FUNCTION_BLOCK UDINT_Param
VAR_INPUT PERSISTENT
	val			: UDINT;
END_VAR

END_FUNCTION_BLOCK

(* stored: Version 1.1.0.1
   POU UDINT_Param: Id {ad9808ce-25ce-489a-8ce0-4c21fc2cde93}, SpecialFunc None *)
